// TIA Portal V19 export
TYPE "LAF_typeGlobalClockMem"
TITLE = Stucture Clock memory byte / Struktur Taktmerker Byte
// Time cycles of clock memory byte. / Zeittakte des Taktmerker Byte
// stored: Access Published
   STRUCT
      cycle100Msec { ExternalAccessible := 'False'; ExternalVisible := 'False'; ExternalWritable := 'False'} : Bool;   // Time cycle 100ms / Zeittakt 100ms
      cycle200Msec { ExternalAccessible := 'False'; ExternalVisible := 'False'; ExternalWritable := 'False'} : Bool;   // Time cycle 200ms / Zeittakt 200ms
      cycle400Msec { ExternalAccessible := 'False'; ExternalVisible := 'False'; ExternalWritable := 'False'} : Bool;   // Time cycle 400ms / Zeittakt 400ms
      cycle500Msec { ExternalAccessible := 'False'; ExternalVisible := 'False'; ExternalWritable := 'False'} : Bool;   // Time cycle 500ms / Zeittakt 500ms
      cycle800Msec { ExternalAccessible := 'False'; ExternalVisible := 'False'; ExternalWritable := 'False'} : Bool;   // Time cycle 800ms / Zeittakt 800ms
      cycle1000Msec { ExternalAccessible := 'False'; ExternalVisible := 'False'; ExternalWritable := 'False'} : Bool;   // Time cycle 1,0sec / Zeittakt 1,0sec
      cycle1600Msec { ExternalAccessible := 'False'; ExternalVisible := 'False'; ExternalWritable := 'False'} : Bool;   // Time cycle 1,6sec / Zeittakt 1,6sec
      cycle2000Msec { ExternalAccessible := 'False'; ExternalVisible := 'False'; ExternalWritable := 'False'} : Bool;   // Time cycle 2,0sec / Zeittakt 2,0sec
   END_STRUCT;
END_TYPE
